FUNCTION F_Convert10V2Temp2 : INT
VAR_INPUT
	i_Value			:	INT;
END_VAR
VAR_OUTPUT
END_VAR
VAR
	r_converted2V 	: 	REAL;
	i_finalValue	:	INT;
END_VAR

// For Convertion of 0-10V Signal from -30 to +70°C

r_converted2V := i_Value * 0.0030518509476;

i_finalValue := REAL_TO_INT((r_converted2V) * 10);

i_finalValue := i_finalValue - (30 * 10); // 0 = -30°

F_Convert10V2Temp2 := i_finalValue;

END_FUNCTION

(* stored: Version 1.1.0.1, ProductVersion 3.1.4024.4
   POU F_Convert10V2Temp2: Id {d30e7e15-2334-4da5-81bb-5e60ecb13a98}, SpecialFunc None *)
